// TIA Portal V18 export
// export: Created 2026-06-16T05:09:47.0620127Z, ExportSetting WithDefaults, DisplayName Totally Integrated Automation Portal, DisplayVersion V18 Update 5, DisplayName TIA Portal Openness, DisplayVersion V18 Update 5, DisplayName TIA Portal Version Control Interface, DisplayVersion V18, DisplayName SINAMICS Startdrive Advanced, DisplayVersion V18 SP2 Update 1, DisplayName SINAMICS Startdrive G110M, G120, G120C, G120D, G120P, G115D, DisplayVersion V18 SP2 Update 1, DisplayName SINAMICS Startdrive G130, G150, S120, S150, SINAMICS MV, S210, G220, S200, DisplayVersion V18 SP2 Update 1, DisplayName STEP 7 Professional, DisplayVersion V18 Update 5, DisplayName STEP 7 Safety, DisplayVersion V18, DisplayName WinCC Advanced / Unified PC, DisplayVersion V18 Update 5
FUNCTION "03_Zone Cumulative" : Void   // FC19, F_FBD
TITLE = AND blocks with one output
{ S7_Optimized_Access := 'TRUE' }
VERSION : 0.1
// v1.0 First Emission
// stored: AutoNumber true, IsIECCheckEnabled false, UDAEnableTagReadback false
BEGIN

REGION Network 1: AREA 1 PB - AREA 1 (Sorter)
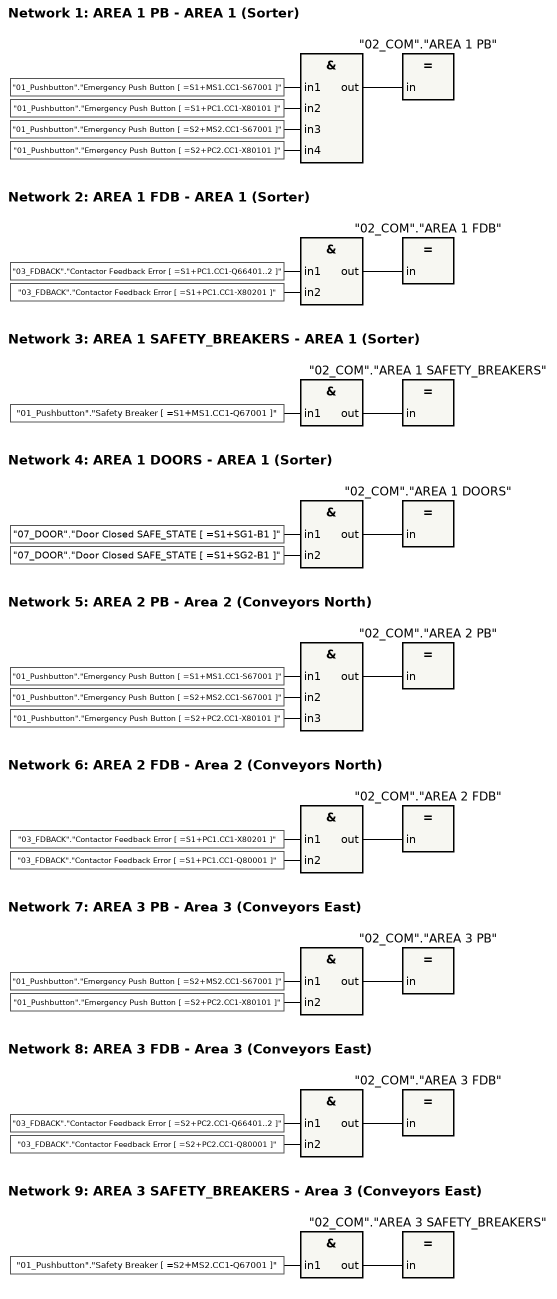
   "02_COM"."AREA 1 PB" := "01_Pushbutton"."Emergency Push Button [ =S1+MS1.CC1-S67001 ]" AND "01_Pushbutton"."Emergency Push Button [ =S1+PC1.CC1-X80101 ]" AND "01_Pushbutton"."Emergency Push Button [ =S2+MS2.CC1-S67001 ]" AND "01_Pushbutton"."Emergency Push Button [ =S2+PC2.CC1-X80101 ]";
END_REGION

REGION Network 2: AREA 1 FDB - AREA 1 (Sorter)
   "02_COM"."AREA 1 FDB" := "03_FDBACK"."Contactor Feedback Error [ =S1+PC1.CC1-Q66401..2 ]" AND "03_FDBACK"."Contactor Feedback Error [ =S1+PC1.CC1-X80201 ]";
END_REGION

REGION Network 3: AREA 1 SAFETY_BREAKERS - AREA 1 (Sorter)
   "02_COM"."AREA 1 SAFETY_BREAKERS" := "01_Pushbutton"."Safety Breaker [ =S1+MS1.CC1-Q67001 ]";
END_REGION

REGION Network 4: AREA 1 DOORS - AREA 1 (Sorter)
   "02_COM"."AREA 1 DOORS" := "07_DOOR"."Door Closed SAFE_STATE [ =S1+SG1-B1 ]" AND "07_DOOR"."Door Closed SAFE_STATE [ =S1+SG2-B1 ]";
END_REGION

REGION Network 5: AREA 2 PB - Area 2 (Conveyors North)
   "02_COM"."AREA 2 PB" := "01_Pushbutton"."Emergency Push Button [ =S1+MS1.CC1-S67001 ]" AND "01_Pushbutton"."Emergency Push Button [ =S2+MS2.CC1-S67001 ]" AND "01_Pushbutton"."Emergency Push Button [ =S2+PC2.CC1-X80101 ]";
END_REGION

REGION Network 6: AREA 2 FDB - Area 2 (Conveyors North)
   "02_COM"."AREA 2 FDB" := "03_FDBACK"."Contactor Feedback Error [ =S1+PC1.CC1-X80201 ]" AND "03_FDBACK"."Contactor Feedback Error [ =S1+PC1.CC1-Q80001 ]";
END_REGION

REGION Network 7: AREA 3 PB - Area 3 (Conveyors East)
   "02_COM"."AREA 3 PB" := "01_Pushbutton"."Emergency Push Button [ =S2+MS2.CC1-S67001 ]" AND "01_Pushbutton"."Emergency Push Button [ =S2+PC2.CC1-X80101 ]";
END_REGION

REGION Network 8: AREA 3 FDB - Area 3 (Conveyors East)
   "02_COM"."AREA 3 FDB" := "03_FDBACK"."Contactor Feedback Error [ =S2+PC2.CC1-Q66401..2 ]" AND "03_FDBACK"."Contactor Feedback Error [ =S2+PC2.CC1-Q80001 ]";
END_REGION

REGION Network 9: AREA 3 SAFETY_BREAKERS - Area 3 (Conveyors East)
   "02_COM"."AREA 3 SAFETY_BREAKERS" := "01_Pushbutton"."Safety Breaker [ =S2+MS2.CC1-Q67001 ]";
END_REGION

REGION Network 10: AREA 3 DOORS - Area 3 (Conveyors East)
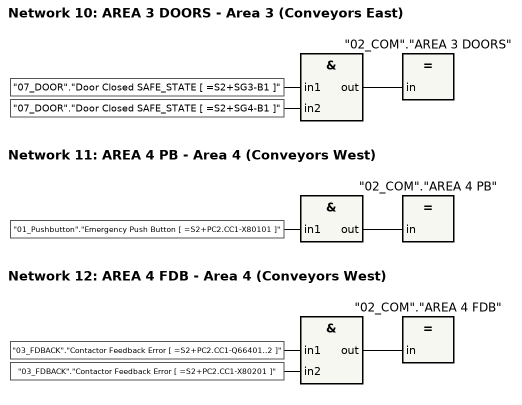
   "02_COM"."AREA 3 DOORS" := "07_DOOR"."Door Closed SAFE_STATE [ =S2+SG3-B1 ]" AND "07_DOOR"."Door Closed SAFE_STATE [ =S2+SG4-B1 ]";
END_REGION

REGION Network 11: AREA 4 PB - Area 4 (Conveyors West)
   "02_COM"."AREA 4 PB" := "01_Pushbutton"."Emergency Push Button [ =S2+PC2.CC1-X80101 ]";
END_REGION

REGION Network 12: AREA 4 FDB - Area 4 (Conveyors West)
   "02_COM"."AREA 4 FDB" := "03_FDBACK"."Contactor Feedback Error [ =S2+PC2.CC1-Q66401..2 ]" AND "03_FDBACK"."Contactor Feedback Error [ =S2+PC2.CC1-X80201 ]";
END_REGION
END_FUNCTION
